FUNCTION f_RobotPtTengelytolTavol : BOOL

f_RobotPtTengelytolTavol:=(GVL.stRobotStatusz.rX<-1.0) OR (GVL.stRobotStatusz.rZ>-111.0);

END_FUNCTION

(* stored: Version 1.1.0.1, ProductVersion 3.1.4020.3
   POU f_RobotPtTengelytolTavol: Id {53f74da6-8f20-48c4-96d2-2e71f627c788}, SpecialFunc None *)
